// TIA Portal project "apples" (V16)

(* hardware
DEVICE "HMI_1"  KTP700 Basic DP
   slot 0: "HMI_1"  KTP700 Basic DP  6AV2 123-2GA03-0AX0  16.0.0.0
   slot 1: "HMI_RT_1"  KTP700 Basic DP  6AV2 123-2GA03-0AX0  16.0.0.0
   slot 7: "HMI_1.MPI/DP_CP_1"  MPI/DP Interface  16.0.0.0
DEVICE "S7300/ET200M station_1"  S7-300 station
   slot 0: "Rail_0"  Rail  6ES7 390-1***0-0AA0
   slot 2: "PLC_1"  CPU 314C-2 DP  6ES7 314-6CH04-0AB0  V3.3
      slot 0: "MPI interface_1"  MPI
      slot 1: "DP interface_1"  DP
      slot 2: "DI 24/DO 16_1"  DI24/DO16
      slot 3: "AI 5/AO 2_1"  AI5/AO2
      slot 4: "Count_1"  Counter
      slot 5: "Positioning_1"  Positioning
*)

// ===== PLC "PLC_1"  CPU 314C-2 DP =====

VAR_GLOBAL   // PLC tag table "Default tag table"
   "Start" AT %M0.0 : Bool;
   "Stop" AT %M0.1 : Bool;
   "box conveyer" AT %Q0.0 : Bool;
   "apple conveyer" AT %Q0.1 : Bool;
   "reset" AT %Q0.2 : Bool;
   "counter" AT %C0 : Counter;
   "box sensor" AT %M0.2 : Bool;
   "apple sensor" AT %M0.3 : Bool;
   "counter output" AT %MW0 : Int;
   "motors" AT %Q0.3 : Bool;
   "restart" AT %Q0.4 : Bool;
END_VAR

ORGANIZATION_BLOCK "Main"   // OB1, LAD
TITLE = "Main Program Sweep (Cycle)"
{ S7_Optimized_Access := 'FALSE' }
VERSION : 0.1
   VAR_TEMP
      OB1_EV_CLASS : Byte;   // Bits 0-3 = 1 (Coming event), Bits 4-7 = 1 (Event class 1)
      OB1_SCAN_1 : Byte;   // 1 (Cold restart scan 1 of OB 1), 3 (Scan 2-n of OB 1)
      OB1_PRIORITY : Byte;   // Priority of OB Execution
      OB1_OB_NUMBR : Byte;   // 1 (Organization block 1, OB1)
      OB1_RESERVED_1 : Byte;   // Reserved for system
      OB1_RESERVED_2 : Byte;   // Reserved for system
      OB1_PREV_CYCLE : Int;   // Cycle time of previous OB1 scan (milliseconds)
      OB1_MIN_CYCLE : Int;   // Minimum cycle time of OB1 (milliseconds)
      OB1_MAX_CYCLE : Int;   // Maximum cycle time of OB1 (milliseconds)
      OB1_DATE_TIME : Date_And_Time;   // Date and time OB1 started
   END_VAR
BEGIN

REGION Network 1
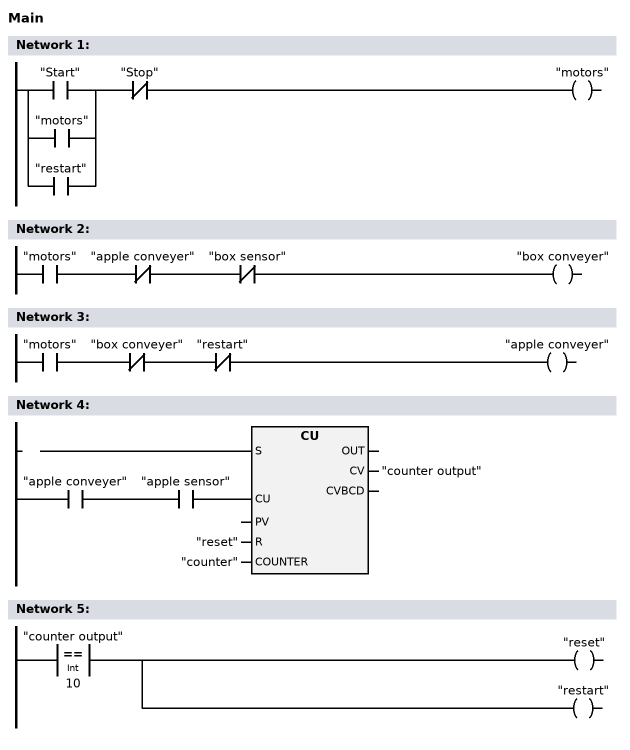
   RUNG wire#powerrail
      Contact( "Start" )
      wire#w1
      I_Contact( "Stop" )
      Coil( "motors" )
   END_RUNG
   RUNG wire#powerrail
      Contact( "motors" )
   END_RUNG wire#w1
   RUNG wire#powerrail
      Contact( "restart" )
   END_RUNG wire#w1
   // the same network as SCL:
   "motors" := ("Start" OR "motors" OR "restart") AND NOT "Stop";
END_REGION

REGION Network 2
   RUNG wire#powerrail
      Contact( "motors" )
      I_Contact( "apple conveyer" )
      I_Contact( "box sensor" )
      Coil( "box conveyer" )
   END_RUNG
   // the same network as SCL:
   "box conveyer" := "motors" AND NOT "apple conveyer" AND NOT "box sensor";
END_REGION

REGION Network 3
   RUNG wire#powerrail
      Contact( "motors" )
      I_Contact( "box conveyer" )
      I_Contact( "restart" )
      Coil( "apple conveyer" )
   END_RUNG
   // the same network as SCL:
   "apple conveyer" := "motors" AND NOT "box conveyer" AND NOT "restart";
END_REGION

REGION Network 4
   // no SCL statement known for Cu: written as a call
   Cu(cu := "apple conveyer" AND "apple sensor", r := "reset", "counter" := "counter", cv => "counter output");
END_REGION

REGION Network 5
   RUNG wire#powerrail
      { S7_Templates := "SrcType := Int" } EQ_Contact(in1 := "counter output", in2 := 10)
      wire#w1
      Coil( "reset" )
   END_RUNG
   RUNG wire#w1
      Coil( "restart" )
   END_RUNG
   // the same network as SCL:
   "reset" := "counter output" = 10;
   "restart" := "reset";
END_REGION
END_ORGANIZATION_BLOCK

(* ===== HMI "HMI_RT_1" =====
system functions are stored by id; their names below are inferred from use

HMI tags "Default tag table"
   "Tag_ScreenNumber" : UInt, internal
   "Move" : Int, internal

Template "Template_1" 800x480
   Button "Exit" at 714,429 size 71x50; TextOff 'Exit'; PictureOff "ExitRuntime_KTP700_Basic_DP_TR"; PictureOn "ExitRuntime_KTP700_Basic_DP_TR"
      on Release: StopRuntime(0)
   Button "Template_Button" at 614,429 size 71x50; TextOff 'Text'
   Button "Template_Button_1" at 514,429 size 71x50; TextOff 'Text'
   Button "Template_Button_2" at 414,429 size 71x50; TextOff 'Text'
   Button "Template_Button_3" at 314,429 size 71x50; TextOff 'Text'
   Button "Template_Button_4" at 214,429 size 71x50; TextOff 'Text'
   Button "Alarms" at 114,429 size 71x50; TextOff 'Alarms'; PictureOff "AlarmDisplay_KTP700_Basic_DP_TR"; PictureOn "AlarmDisplay_KTP700_Basic_DP_TR"
      on Release: function_ef3f5d25("Alarm window_Unacknowledged", -1)
   Button "Start screen" at 14,429 size 71x50; TextOff 'Start screen'; PictureOff "NavigateHome_KTP700_Basic_DP_TR"; PictureOn "NavigateHome_KTP700_Basic_DP_TR"
      on Release: ActivateScreen("Root screen", 0)
   SymbolicIOField "Symbolic_IO_Field_Screen" at 93,9 size 600x33; TextOff '0'; TextOn '1'; TextList "TextList_ScreenNames"
      ProcessValue <- "Tag_ScreenNumber"
      on Change: ActivateScreenByNumber("Tag_ScreenNumber", 0)
   DateTimeField "HmiScreenItemData" at 695,25 size 105x25
   DateTimeField "HmiScreenItemData_1" at 695,0 size 105x25
   GraphicView "Logo" at 0,0 size 91x51; Picture "Logo of HMI_1"

screen "Root screen" 800x480, template "Template_1"
   on GenerateScreen: SetTag("Tag_ScreenNumber", 1); function_f9c01323("Move", 1, 100, 0, 1)
   Button "Button_1" at 53,87 size 96x36; TextOff 'Start'
   Button "Button_2" at 52,140 size 96x32; TextOff 'Stop'
   IOField "I/O field_1" at 570,54 size 96x32; FormatPattern 9999999
   GraphicView "Graphic view_1" at 20,301 size 600x76; Picture "Graphic_1"
   GraphicView "Graphic view_2" at 555,105 size 216x137; Picture "Graphic_2"
   GraphicView "Graphic view_3" at 705,171 size 85x53; Picture "Graphic_3"
   GraphicView "Graphic view_4" at 33,376 size 84x53; Picture "Graphic_3"
   GraphicView "Graphic view_5" at 454,197 size 43x56; Picture "Graphic_4"
   GraphicView "Graphic view_6" at 557,103 size 41x68; Picture "Graphic_5"
   GraphicView "Graphic view_7" at 68,247 size 88x90; Picture "Graphic_6"
   GraphicView "Graphic view_8" at 673,87 size 53x47; Picture "apple"
      DiagonalMovement <- "Move"
      Visibility <- "Move"
*)